PROGRAM DerotatorControl
VAR_INPUT
	enable:		BOOL;
	reset:		BOOL;
	left:		BOOL;
	right:		BOOL;
	position:	LREAL;
END_VAR
VAR_OUTPUT
	Error:		BOOL;
	ErrorID:	UDINT;
	actual_position:	LREAL;
END_VAR
VAR
	// move to given position
	MoveAxis: 			BOOL;
	// calibrate the axis
	HomeAxis:			BOOL;

	DerotatorAxis:	FB_Axis2;
	DerotatorEvent:	FB_EventLog;
END_VAR
VAR CONSTANT
	// current position of the calibration cam. Apply an offset here if necessary
	calibration_position:	LREAL := 0.0;
END_VAR

// TODO: Limit switch for Derotator axis!

(*
Homing in Endlage über die Probe Unit:

https://infosys.beckhoff.com/index.php?content=../content/1031/ax5000_usermanual/html/ax5000_homing_hardware_end_position.htm&id=12221
*)
enable := TelescopeControl.power OR PendantControl.Derotator_enable;

DeRotatorAxis(
	enable := 			enable,
	Reset := 			Reset,
	MoveAxis :=			MoveAxis,
	HomeAxis :=			HomeAxis,
	Position := 		position, 
	Enable_Positive := 	TRUE,
	Enable_Negative := 	TRUE,
	Jog_Forward := 		right,
	Jog_Backwards := 	left,
	bCalibrationCam :=	FALSE,	// TODO: place limit switch from DIO here
	isModuloAxis :=		TRUE,
	ActualPosition => 	actual_position,
	Error => 			Error,
	ErrorID => 			ErrorID,
	AxisRef :=			GVL_Telescope.DerotatorAxisRef);
	
IF DeRotatorAxis.MoveDone THEN
	MoveAxis := FALSE;
END_IF

IF DeRotatorAxis.HomeDone THEN
	HomeAxis := FALSE;
END_IF
	
IF DeRotatorAxis.ResetDone THEN
	reset := FALSE;
END_IF

DerotatorEvent(	
	Trigger := 		Error, 
	Level := 		ADSLOG_MSGTYPE_ERROR,
	FormatString :=	'Derotator Axis Error: %s',
	OnMessage := 	DWORD_TO_HEXSTR(ErrorID, 4, FALSE),
	OffMEssage := 	'OK',
	OffLevel := 	ADSLOG_MSGTYPE_HINT);

END_PROGRAM

(* stored: Version 1.1.0.1, ProductVersion 3.1.4024.6
   POU DerotatorControl: Id {75f3d994-c6e1-4455-a5dc-0a32056448e8}, SpecialFunc None *)
